// TIA Portal V21 export
FUNCTION_BLOCK "FB607"   // FB607, LAD
TITLE = FB607
{ S7_Optimized_Access := 'FALSE' }
AUTHOR : PRECISE
FAMILY : PRECISE
// CIP MIXING
// stored: AutoNumber false, SetENOAutomatically false
   VAR_INPUT
      CipSelected : Bool;
      CycleEnable : Bool;
      CycleRunning : Bool;
      SecPulse : Bool;
      AlwaysTrue : Bool;
      MixingTimeBaseSel : Bool;   // 0 - secs, 1 - mins
      SetTimeMins : Int := 30;
      SetTimeSecs : Int;
      ActualRepetition : Int;
   END_VAR
   VAR_OUTPUT
      Started : Bool;
      Mixer : Bool;   // Pump Casing Drain
      TimeMinsPv : DInt;
      TimeSecsPv : DInt;
      StepStatus : String[60];
      Print : "MixingPrint";
   END_VAR
   VAR_IN_OUT
      Over : Bool;
   END_VAR
   VAR
      RE1 : Bool;
      RE2 : Bool;
      RE3 : Bool;
      MixingTimer { S7_SetPoint := 'True'} : "FB101";
   END_VAR
   VAR_TEMP   // added for the SCL form of the ladder/FBD networks
      _w1 : Bool;
   END_VAR
BEGIN

REGION Network 1: MixingStarted
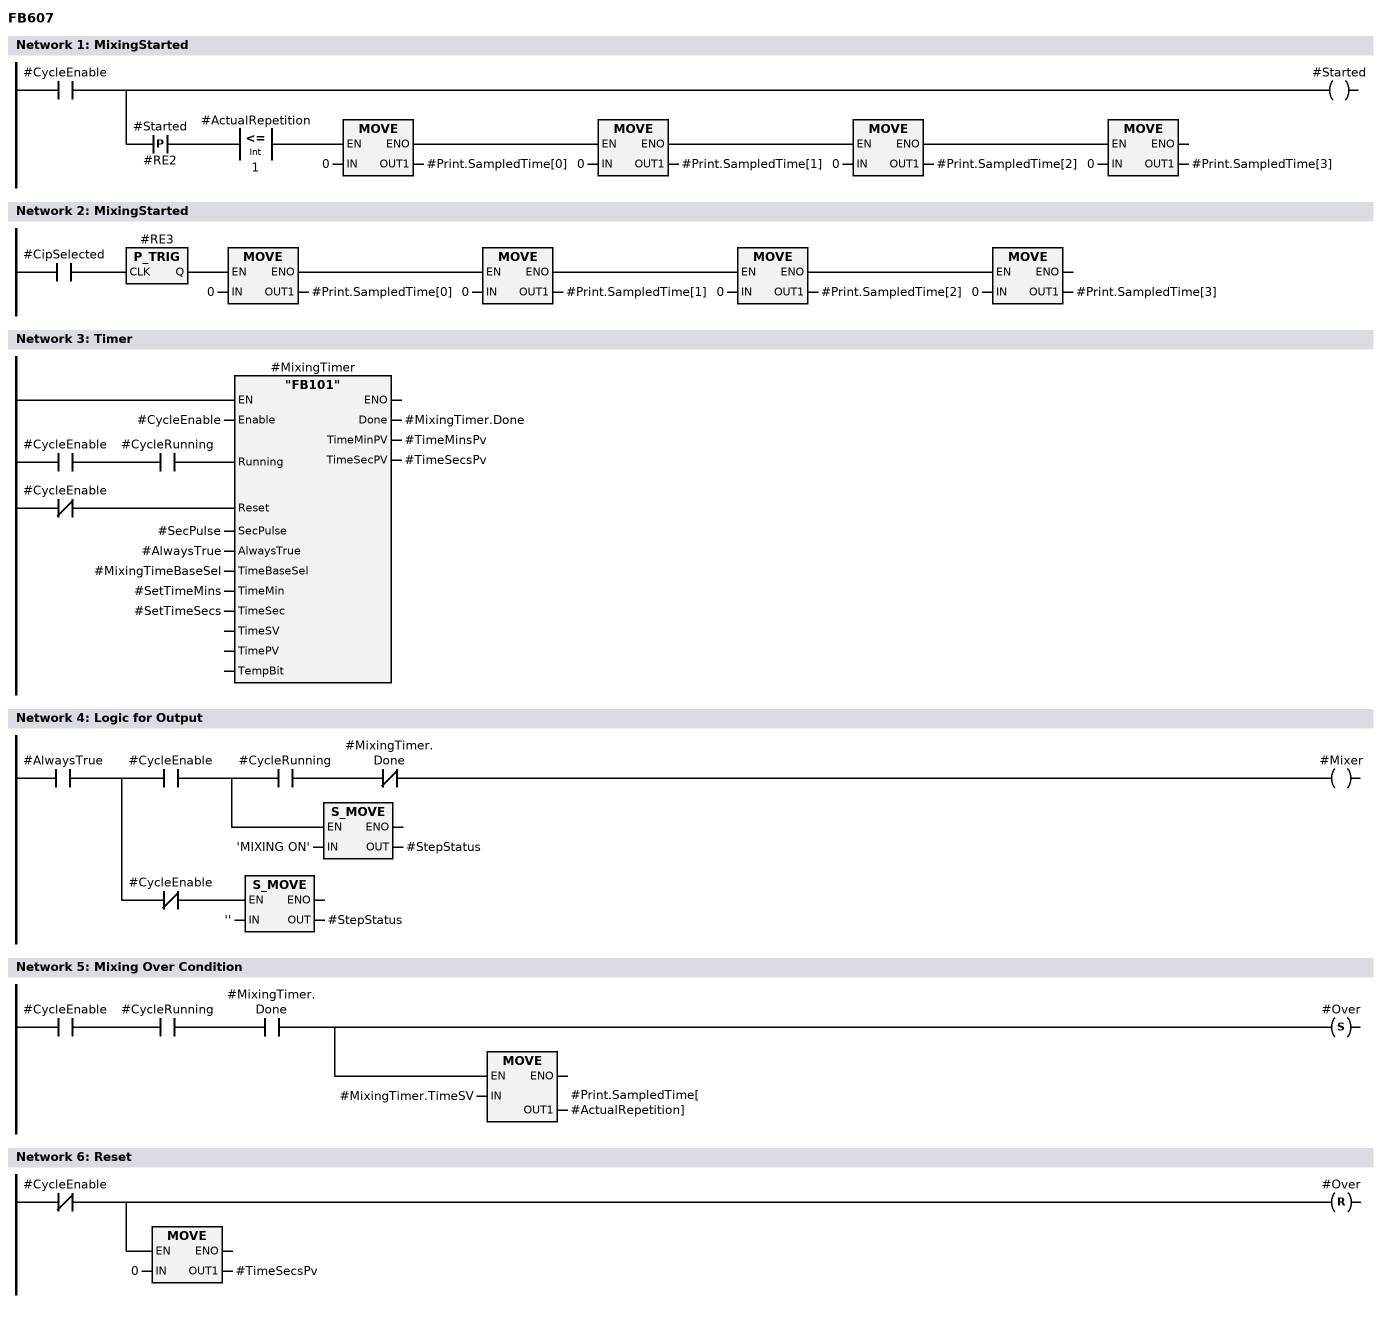
   RUNG wire#powerrail
      Contact( #CycleEnable )
      wire#w1
      Coil( #Started )
   END_RUNG
   RUNG wire#w1
      P_Contact(operand := #Started, bit := #RE2)
      { S7_Templates := "SrcType := Int" } LE_Contact(in1 := #ActualRepetition, in2 := 1)
      Move(in := 0, out1 => #Print.SampledTime[0])
      Move(in := 0, out1 => #Print.SampledTime[1])
      Move(in := 0, out1 => #Print.SampledTime[2])
      Move(in := 0, out1 => #Print.SampledTime[3])
   END_RUNG
   // the same network as SCL:
   #Started := #CycleEnable;
   #_w1 := #CycleEnable AND #Started AND NOT #RE2;   // rising edge of #Started
   #RE2 := #Started;
   IF #_w1 AND (#ActualRepetition <= 1) THEN
       #Print.SampledTime[0] := 0;
       #Print.SampledTime[1] := 0;
       #Print.SampledTime[2] := 0;
       #Print.SampledTime[3] := 0;
   END_IF;
END_REGION

REGION Network 2: MixingStarted
   RUNG wire#powerrail
      Contact( #CipSelected )
      P_Trig( #RE3 )
      Move(in := 0, out1 => #Print.SampledTime[0])
      Move(in := 0, out1 => #Print.SampledTime[1])
      Move(in := 0, out1 => #Print.SampledTime[2])
      Move(in := 0, out1 => #Print.SampledTime[3])
   END_RUNG
   // the same network as SCL:
   #_w1 := #CipSelected AND NOT #RE3;   // rising edge
   #RE3 := #CipSelected;
   IF #_w1 THEN
       #Print.SampledTime[0] := 0;
       #Print.SampledTime[1] := 0;
       #Print.SampledTime[2] := 0;
       #Print.SampledTime[3] := 0;
   END_IF;
END_REGION

REGION Network 3: Timer
   RUNG wire#powerrail
      #MixingTimer(Running := wire#w1, Reset := wire#w2, Enable := #CycleEnable, SecPulse := #SecPulse, AlwaysTrue := #AlwaysTrue, TimeBaseSel := #MixingTimeBaseSel, TimeMin := #SetTimeMins, TimeSec := #SetTimeSecs, TimeSV :=, TimePV :=, TempBit :=, Done => #MixingTimer.Done, TimeMinPV => #TimeMinsPv, TimeSecPV => #TimeSecsPv)
   END_RUNG
   RUNG wire#powerrail
      Contact( #CycleEnable )
      Contact( #CycleRunning )
   END_RUNG wire#w1
   RUNG wire#powerrail
      I_Contact( #CycleEnable )
   END_RUNG wire#w2
   // the same network as SCL:
   #MixingTimer(Enable := #CycleEnable,   // "FB101"
                Running := #CycleEnable AND #CycleRunning,
                Reset := NOT #CycleEnable,
                SecPulse := #SecPulse,
                AlwaysTrue := #AlwaysTrue,
                TimeBaseSel := #MixingTimeBaseSel,
                TimeMin := #SetTimeMins,
                TimeSec := #SetTimeSecs,
                Done => #MixingTimer.Done,
                TimeMinPV => #TimeMinsPv,
                TimeSecPV => #TimeSecsPv);
END_REGION

REGION Network 4: Logic for Output
   RUNG wire#powerrail
      Contact( #AlwaysTrue )
      wire#w1
      Contact( #CycleEnable )
      wire#w2
      Contact( #CycleRunning )
      I_Contact( #MixingTimer.Done )
      Coil( #Mixer )
   END_RUNG
   RUNG wire#w2
      S_Move(in := 'MIXING ON', out => #StepStatus)
   END_RUNG
   RUNG wire#w1
      I_Contact( #CycleEnable )
      S_Move(in := '', out => #StepStatus)
   END_RUNG
   // the same network as SCL:
   #_w1 := #AlwaysTrue AND #CycleEnable;
   #Mixer := #_w1 AND #CycleRunning AND NOT #MixingTimer.Done;
   IF #_w1 THEN #StepStatus := 'MIXING ON'; END_IF;
   IF #AlwaysTrue AND NOT #CycleEnable THEN #StepStatus := ''; END_IF;
END_REGION

REGION Network 5: Mixing Over Condition
   RUNG wire#powerrail
      Contact( #CycleEnable )
      Contact( #CycleRunning )
      Contact( #MixingTimer.Done )
      wire#w1
      S_Coil( #Over )
   END_RUNG
   RUNG wire#w1
      Move(in := #MixingTimer.TimeSV, out1 => #Print.SampledTime[#ActualRepetition])
   END_RUNG
   // the same network as SCL:
   IF #CycleEnable AND #CycleRunning AND #MixingTimer.Done THEN
       #Over := TRUE;
       #Print.SampledTime[#ActualRepetition] := #MixingTimer.TimeSV;
   END_IF;
END_REGION

REGION Network 6: Reset
   RUNG wire#powerrail
      I_Contact( #CycleEnable )
      wire#w1
      R_Coil( #Over )
   END_RUNG
   RUNG wire#w1
      { S7_GenerateENO := "TRUE" } Move(in := 0, out1 => #TimeSecsPv)
   END_RUNG
   // the same network as SCL:
   IF NOT #CycleEnable THEN
       #Over := FALSE;
       #TimeSecsPv := 0;
   END_IF;
END_REGION
END_FUNCTION_BLOCK
